{attribute 'GeneratedUsingTerminal: EL3011-0000-0016'}
{attribute addProperty BoxType "EL3011-0000-0016"}
{attribute addProperty Id "AI_StandardAT %I*AI_Standard_Channel_4A3944819WcStateAT %I*WcState_9091E0EB2InfoDataAT %I*InfoData_94A18F5E2"}
{attribute addProperty CRC "1943597556"}
{attribute addProperty Size "13"}
TYPE EL3011_73D8F1F4 EXTENDS EtcSlaveTerminalBase_947E5A46 :
STRUCT
	{attribute addProperty Name "AI_Standard"}
	AI_Standard : AI_Standard_Channel_4A394481;
	{attribute addProperty Name "WcState"}
	WcState : WcState_9091E0EB;
	{attribute addProperty Name "InfoData"}
	InfoData : InfoData_94A18F5E;
END_STRUCT
END_TYPE

(* stored: Version 1.2.0.0, ProductVersion 3.1.4024.9
   DUT EL3011_73D8F1F4: Id {0f4903e6-68c7-48c1-98f8-0c4d19b1344e} *)
